(* CODESYS project SILO.project

Project tree, tasks and I/O mapping:
  Device : CODESYS Control Win V3, 3S - Smart Software Solutions GmbH, order no. 305021, version 3.5.11.30
    application Application
      libraries: Standard, * (System)
      task MainTask (cyclic, interval t#20ms, priority 1) calls PLC_PRG
      program PLC_PRG [LD]
*)

// Device/Application/PLC_PRG
PROGRAM PLC_PRG
VAR
	START : BOOL;
	STOP : BOOL;
	P1: BOOL;
	P2: BOOL;
	EVAL: BOOL;
	TOF_1: TOF;
	ET1: TIME;
	TON_1: TON;
	ET2: TIME;
	P3: BOOL;
	AUX1: BOOL;
	AUX2: BOOL;
END_VAR
VAR // added by the converter: edge detectors and wires of the graphical bodies
    _rt1, _rt2 : R_TRIG;
END_VAR

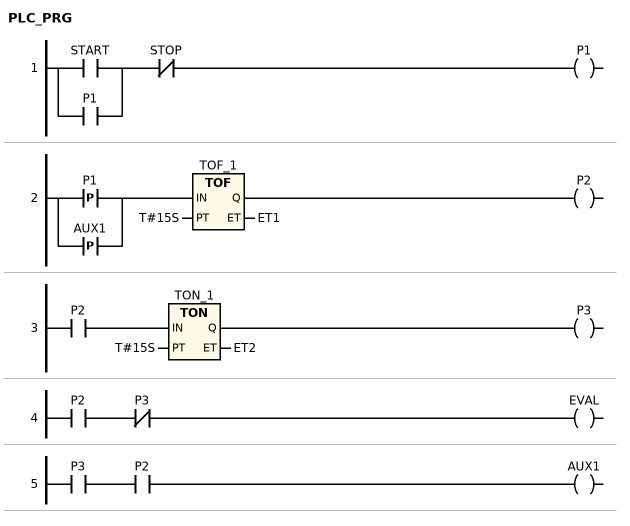
// NETWORK 1
P1 := (START OR P1) AND NOT STOP;

// NETWORK 2
_rt1(CLK := P1);
_rt2(CLK := AUX1);
TOF_1(IN := _rt1.Q OR _rt2.Q, PT := T#15S, ET => ET1); // TOF
P2 := TOF_1.Q;

// NETWORK 3
TON_1(IN := P2, PT := T#15S, ET => ET2); // TON
P3 := TON_1.Q;

// NETWORK 4
EVAL := P2 AND NOT P3;

// NETWORK 5
AUX1 := P3 AND P2;

END_PROGRAM
